PROGRAM PRG_GEM2_DIFF_PUMP
VAR
END_VAR

(*Gauges*)
DSG_PIN(sNetId:='172.21.88.138.1.1' , nPort:=851 , sVarName:='GVL_Devices.AT2L0_SOLID_PIN_01',iWatchdog:=Main.iWatchdog,IG=> ); // Downstream Gauge from Down Stream PLC System
(*EM2L0*)
GEM2_GPI_30(PG=>);
GEM2_GCC_30(PG:=GEM2_GPI_30.PG,IG=>);
GEM2_GPI_31(PG=>);
GEM2_GPI_50(PG=>);
GEM2_GCC_50(PG:=GEM2_GPI_50.PG,IG=>);
GEM2_GPI_51(PG=>);
GEM2_GPI_60(PG=>);
GEM2_GCC_60(PG:=GEM2_GPI_60.PG,IG=>);
GEM2_GPI_61(PG=>);
GEM2_GPI_70(PG=>);
GEM2_GCC_70(PG:=GEM2_GPI_70.PG,IG=>);

(*VALVES*)
(*Aperture valve may open when Detector and Attenuator N2 valves are closed. Override provided *)
 (* to Include PMPS ILK with the EXTILK bit*)
(*apperture valves*)
GEM2_VGC_10(i_stUSG := GEM2_GPI_10.PG, i_stDSG:= GEM2_GPI_10.PG,i_xDis_DPIlk := TRUE, i_xEPS_OK := TRUE,
		i_xPMPS_OK := TRUE, i_xExt_OK := xGEM2_AperturesOpnOK, i_xOverrideMode := xGEM2OverrideMode,i_xReset := xFastFaultReset,io_fbFFHWO :=g_FastFaultOutput1);
GEM2_VGC_20(i_stUSG := GEM2_GPI_10.PG, i_stDSG:= GEM2_GCC_30.IG,i_xDis_DPIlk := TRUE, i_xEPS_OK := TRUE,
		i_xPMPS_OK := TRUE, i_xExt_OK := xGEM2_AperturesOpnOK, i_xOverrideMode := xGEM2OverrideMode,i_xReset := xFastFaultReset,io_fbFFHWO :=g_FastFaultOutput1);
GEM2_VGC_30(i_stUSG := GEM2_GCC_30.IG, i_stDSG:= GEM2_GCC_30.IG,i_xDis_DPIlk := TRUE, i_xEPS_OK := TRUE,
		i_xPMPS_OK := TRUE, i_xExt_OK := xGEM2_AperturesOpnOK, i_xOverrideMode := xGEM2OverrideMode,i_xReset := xFastFaultReset,io_fbFFHWO :=g_FastFaultOutput1);
GEM2_VGC_40(i_stUSG := GEM2_GCC_50.IG, i_stDSG:= GEM2_GCC_50.IG,i_xDis_DPIlk := TRUE, i_xEPS_OK := TRUE,
		i_xPMPS_OK := TRUE, i_xExt_OK := xGEM2_AperturesOpnOK, i_xOverrideMode := xGEM2OverrideMode,i_xReset := xFastFaultReset,io_fbFFHWO :=g_FastFaultOutput1);	
GEM2_VGC_50(i_stUSG := GEM2_GCC_30.IG, i_stDSG:= GEM2_GCC_60.IG,i_xDis_DPIlk := TRUE, i_xEPS_OK := TRUE,
		i_xPMPS_OK := TRUE, i_xExt_OK := xGEM2_AperturesOpnOK, i_xOverrideMode := xGEM2OverrideMode,i_xReset := xFastFaultReset,io_fbFFHWO :=g_FastFaultOutput1);
GEM2_VGC_60(i_stUSG := GEM2_GCC_60.IG, i_stDSG:= GEM2_GCC_70.IG,i_xDis_DPIlk := TRUE, i_xEPS_OK := TRUE,
		i_xPMPS_OK := TRUE, i_xExt_OK := xGEM2_AperturesOpnOK, i_xOverrideMode := xGEM2OverrideMode,i_xReset := xFastFaultReset,io_fbFFHWO :=g_FastFaultOutput1);
(*downstream isolation valve*)
GEM2_VGC_70(i_stUSG := GEM2_GCC_70.IG, i_stDSG:= DSG_PIN.IG,i_xDis_DPIlk := FALSE, i_xEPS_OK := TRUE,
		i_xPMPS_OK := TRUE, i_xExt_OK := TRUE, i_xOverrideMode := xGEM2OverrideMode,i_xReset := xFastFaultReset,io_fbFFHWO :=g_FastFaultOutput1);
DSV_VGC(VGC=>);

(*Turbo vent valves NO*)//Deprecated
GEM2_VVC_30(i_stPTM :=GEM2_PTM_30.iq_stPtm);
GEM2_VVC_50(i_stPTM :=GEM2_PTM_50.iq_stPtm);
GEM2_VVC_70(i_stPTM :=GEM2_PTM_70.iq_stPtm);
(*This part was added to Close all the Turbo's NO vent valves, These valves are capped off, and wont be in use*)
GEM2_VVC_30.M_Close(TRUE);
GEM2_VVC_50.M_Close(TRUE);
GEM2_VVC_70.M_Close(TRUE);


(*Turbo Isolation valves*)
 GEM2_VRC_30(i_xExtILK_OK := F_TurboGateValve_ILK(GEM2_PTM_30.iq_stPtm,GEM2_GPI_30.PG),i_xOverrideMode := xGEM2OverrideMode);
 GEM2_VRC_50(i_xExtILK_OK := F_TurboGateValve_ILK(GEM2_PTM_50.iq_stPtm,GEM2_GPI_50.PG),i_xOverrideMode := xGEM2OverrideMode);
 GEM2_VRC_60(i_xExtILK_OK := F_TurboGateValve_ILK(GEM2_PTM_60.iq_stPtm,GEM2_GPI_60.PG),i_xOverrideMode := xGEM2OverrideMode);
 GEM2_VRC_70(i_xExtILK_OK := F_TurboGateValve_ILK(GEM2_PTM_70.iq_stPtm,GEM2_GPI_70.PG),i_xOverrideMode := xGEM2OverrideMode);

(*Turbo Pumps*)
GEM2_PTM_30(i_xExtILKOK:=F_TurboExtILK_NO(GEM2_PTM_30.iq_stPtm, GEM2_GPI_31.PG,
						GEM2_GPI_30.PG,GEM2_VVC_30.q_stValve,GEM2_PMF_30.iq_stPFO),
		i_stGauge:=GEM2_GPI_31.PG,i_rMaxBackingPressure :=0.6);
GEM2_PTM_50(i_xExtILKOK:=F_TurboExtILK_NO(GEM2_PTM_50.iq_stPtm, GEM2_GPI_51.PG,
						GEM2_GPI_50.PG,GEM2_VVC_50.q_stValve,GEM2_PMF_50.iq_stPFO),
		i_stGauge:=GEM2_GPI_51.PG,i_rMaxBackingPressure :=0.6);
GEM2_PTM_60(i_xExtILKOK:=F_TurboExtILK_NO(GEM2_PTM_60.iq_stPtm, GEM2_GPI_61.PG,
						GEM2_GPI_60.PG,GEM2_VVC_70.q_stValve,GEM2_PMF_60.iq_stPFO),
		i_stGauge:=GEM2_GPI_61.PG,i_rMaxBackingPressure :=0.4);
GEM2_PTM_70(i_xExtILKOK:=F_TurboExtILK_NO(GEM2_PTM_70.iq_stPtm, GEM2_GPI_61.PG,
						GEM2_GPI_70.PG,GEM2_VVC_70.q_stValve,GEM2_PMF_60.iq_stPFO),
		i_stGauge:=GEM2_GPI_61.PG,i_rMaxBackingPressure :=0.4);

(*Roughing pumps*)
GEM2_PMF_30(xExtIlk:= TRUE, TurboIsOn:= GEM2_PTM_30.iq_stPtm.q_RunDO); 
GEM2_PMF_50(xExtIlk:= TRUE, TurboIsOn:= GEM2_PTM_50.iq_stPtm.q_RunDO); 
GEM2_PMF_60(xExtIlk:= TRUE, TurboIsOn:= (GEM2_PTM_60.iq_stPtm.q_RunDO OR GEM2_PTM_70.iq_stPtm.q_RunDO));

END_PROGRAM

(* stored: Version 1.1.0.1, ProductVersion 3.1.4022.18
   POU PRG_GEM2_DIFF_PUMP: Id {851181dd-ec63-4e65-94b1-0ffbf8be6c3d}, SpecialFunc None *)
